PROGRAM PRG_MFuncControl
VAR
	bTestValveOutput		: BOOL;
END_VAR


IF bMFunc[11] THEN
	bTestValveOutput	:= TRUE;
	bQuitMFunc[11]		:= TRUE;
END_IF


IF bMFunc[12] THEN
	bTestValveOutput	:= FALSE;
	bQuitMFunc[12]		:= TRUE;
END_IF

END_PROGRAM

(* stored: Version 1.1.0.1, ProductVersion 3.1.4022.6
   POU PRG_MFuncControl: Id {19677d06-9e27-4323-bf51-bb01aefc8330}, SpecialFunc None *)
